{attribute 'qualified_only'}
TYPE SectionEnum :
(
	NULL_SECTION := -1,
	PAPER,
	CARDBOARD_CORNERGUARD,
	CHIPBOARD,
	WOOD_BUNK,
	OUTPUT,
	
	size
);
END_TYPE

(* stored: Version 1.1.0.1, ProductVersion 3.1.4024.11
   DUT SectionEnum: Id {7c824539-95c8-4ad1-8c1a-2206d5879333} *)
